// TIA Portal V19 export
VAR_GLOBAL   // PLC tag table "Equipment_Template_DefaultTagTable_10"
END_VAR
